(* PLC project test, Неизвестно Unnamed 1 *)
(* stored: creationDateTime 2025-01-15T16:56:00, modificationDateTime 2025-01-16T03:35:33 *)

PROGRAM PLC_PRG
  VAR
    rHysteresis : REAL := 1;
    SR_0 : SR;
  END_VAR
  VAR  (* added by the conversion: wires and edge detectors of the diagram *)
    _ADD4_OUT : ANY;
    _LT12_OUT : BOOL;
    _SUB15_OUT : ANY;
  END_VAR

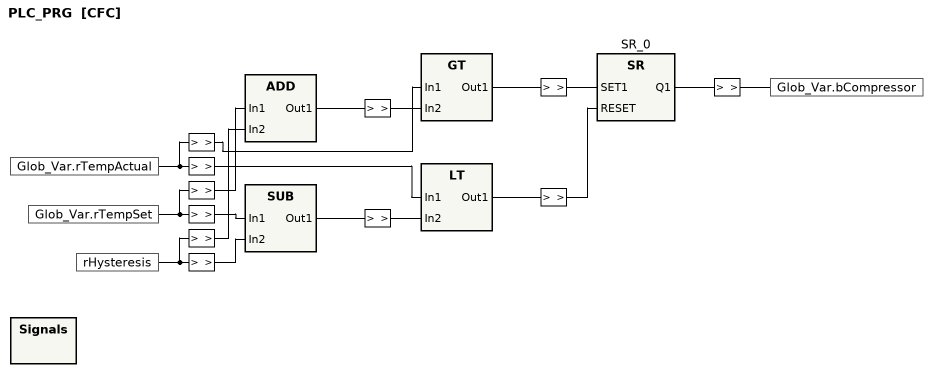
(* CFC diagram, written out as Structured Text *)
SR_0(SET1 := Glob_Var.rTempActual > _ADD4_OUT, RESET := _LT12_OUT);
Glob_Var.bCompressor := SR_0.Q1;
_ADD4_OUT := Glob_Var.rTempSet + rHysteresis;
_LT12_OUT := Glob_Var.rTempActual < _SUB15_OUT;
_SUB15_OUT := Glob_Var.rTempSet - rHysteresis;
Signals();
END_PROGRAM

PROGRAM Signals
  VAR
    TON_0 : TON;
    TON_1 : TON;
    BLINK_0 : BLINK;
    timSignalTime : TIME := TIME#1s0ms;
  END_VAR

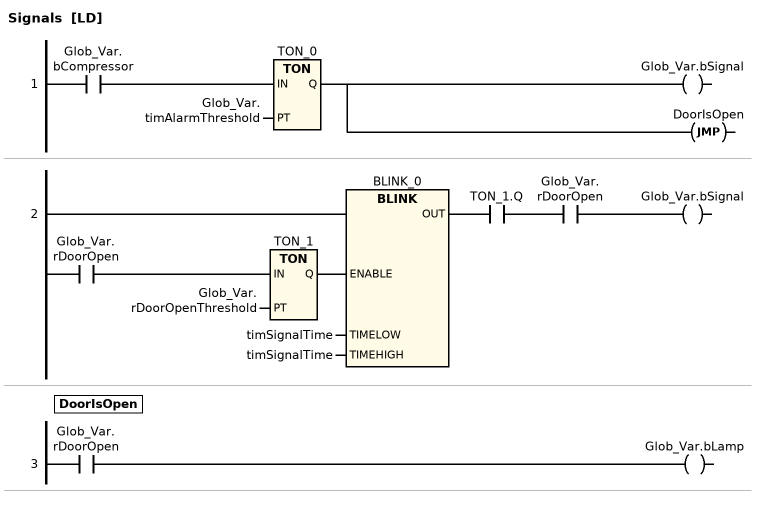
(* LD diagram, written out as Structured Text *)

TON_0(IN := Glob_Var.bCompressor, PT := Glob_Var.timAlarmThreshold);
Glob_Var.bSignal := TON_0.Q;
IF TON_0.Q THEN JMP DoorIsOpen; END_IF;

TON_1(IN := Glob_Var.rDoorOpen, PT := Glob_Var.rDoorOpenThreshold);
BLINK_0(ENABLE := TON_1.Q, TIMELOW := timSignalTime, TIMEHIGH := timSignalTime);
Glob_Var.bSignal := BLINK_0.OUT AND TON_1.Q AND Glob_Var.rDoorOpen;
DoorIsOpen:

Glob_Var.bLamp := Glob_Var.rDoorOpen;
END_PROGRAM

PROGRAM Simulation
  VAR
    T1 : TON;  (* The temperature is decreased on a time delay, when the comepressor has been activated *)
    P_Cooling : TIME := TIME#500ms;
    xReduceTemp : BOOL;  (* Signal for dereasing the temperature *)
    T2 : TON;  (* The temperature is increased on a time delay, when the compressor has been activated *)
    P_Environment : TIME := TIME#2s0ms;  (* Delay time when the door is closed *)
    P_EnvironmentDoorOpen : TIME := TIME#1s0ms;  (* Delay time when the door is open *)
    xRaiseTemp : BOOL;  (* Signal for increasing the temperature *)
    timTemp : TIME;  (* Delay time *)
    iCounter : INT;
  END_VAR

                    iCounter := iCounter+1;     // No function, just for demonstration purposes.

// After the compressor has been activated due to TempActual being too high, the temperature decreases.
// The temperature is decremented by 0.1°C per cycle after a delay of P_Cooling
IF Glob_VAR.bCompressor THEN
    T1(IN:= Glob_Var.bCompressor, PT:= P_Cooling, Q=>xReduceTemp);
    IF xReduceTemp THEN
        Glob_Var.rTempActual := Glob_Var.rTempActual-0.1;
        T1(IN:=FALSE);
    END_IF
END_IF

//If the door is open, the warming occurs faster; SEL selects P_EnvironmentDoorOpen
timTemp:=SEL(Glob_Var.rDoorOpen, P_Environment, P_EnvironmentDoorOpen);

//If the compressor is not in operation, then the cooling chamber becomes warmer.
//The  temperature is incremented by 0.1°C per cycle after a delay of tTemp
T2(IN:= TRUE, PT:= timTemp, Q=>xRaiseTemp);
IF xRaiseTemp THEN
    Glob_Var.rTempActual := Glob_Var.rTempActual + 0.1;
    T2(IN:=FALSE);
END_IF

                  
END_PROGRAM

CONFIGURATION Device
  RESOURCE Application ON PLC
    {attribute 'qualified_only'}
    VAR_GLOBAL  (* Glob_Var *)
      rTempActual : REAL := 8;
      rTempSet : REAL := 8;
      rDoorOpen : BOOL := FALSE;
      timAlarmThreshold : TIME := TIME#30ms;  (* Compressor running time after which a signal sounds *)
      rDoorOpenThreshold : TIME := TIME#10s0ms;  (* Time from opening the door after which a signal should sound *)
      bCompressor : BOOL;
      bSignal : BOOL := FALSE;
      bLamp : BOOL := FALSE;
    END_VAR
    TASK MainTask(INTERVAL := T#20ms, PRIORITY := 0);
    PROGRAM Simulation WITH MainTask : Simulation;
    PROGRAM PLC_PRG WITH MainTask : PLC_PRG;
  END_RESOURCE
  RESOURCE Res0 ON PLC
  END_RESOURCE
END_CONFIGURATION
